{attribute 'GeneratedUsingTerminal: ELX4181-0000-0016'}
{attribute addProperty BoxType "ELX4181-0000-0016"}
{attribute addProperty Id "EtcSlaveTerminalBaseCh_1Ch_1_8C75A2992WcStateAT %I*WcState_0B2B16F91InfoDataAT %I*InfoData_90184F0C16"}
{attribute addProperty CRC "3482863652"}
{attribute addProperty Size "19"}
TYPE ELX4181_CF984824 EXTENDS EtcSlaveTerminalBase :
STRUCT
	{attribute addProperty Name "Ch_1"}
	Ch_1 : Ch_1_8C75A299;
	{attribute addProperty Name "WcState"}
	WcState : WcState_0B2B16F9;
	{attribute addProperty Name "InfoData"}
	InfoData : InfoData_90184F0C;
END_STRUCT
END_TYPE

(* stored: Version 1.2.0.0, ProductVersion 3.1.4024.9
   DUT ELX4181_CF984824: Id {74e8c1a3-6f8d-47be-afc7-06046c042579} *)
